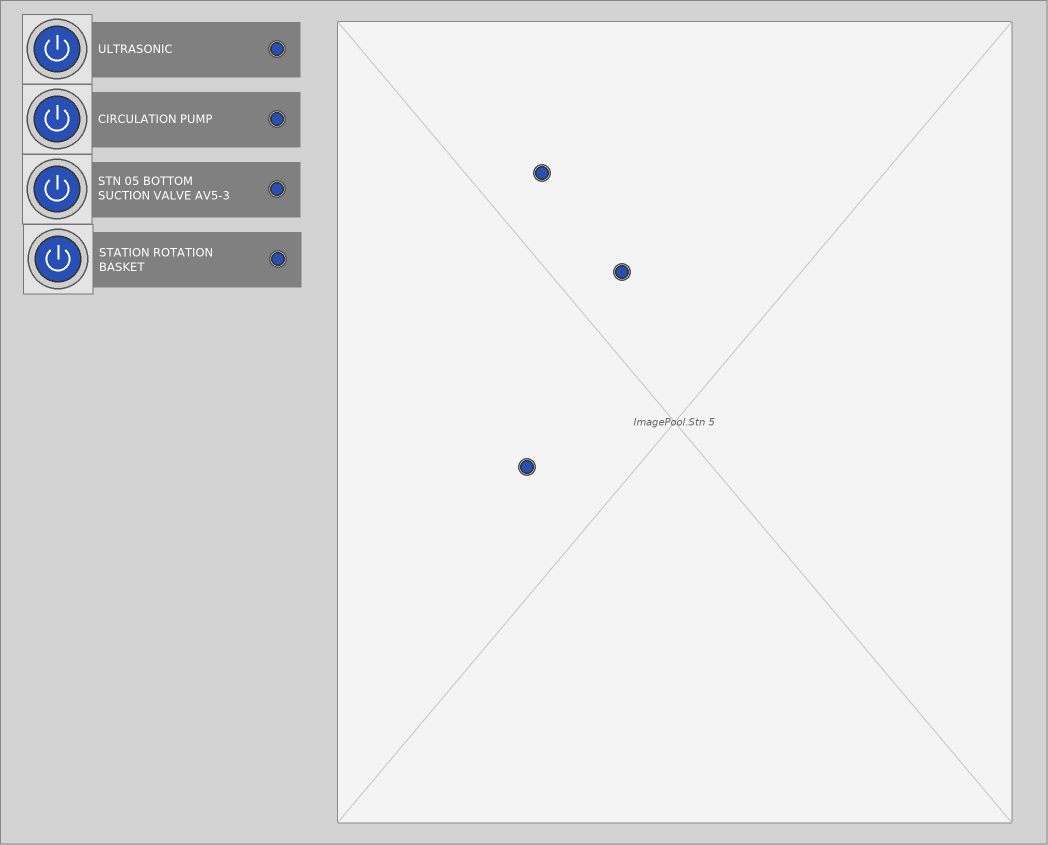
VISUALIZATION Recipe_Station05  // 1048x845
    Rectangle (0,0 1048x845)
    Image (337,21 675x802), image: ImagePool.Stn 5
    RoundedRectangle (61,22 239x55)
    Label (95,41 163x16), "ULTRASONIC"
    Lamp1 (267,39 20x20), variable: DSScrMapSSUR.DsSubRecipeMemory.bOut3EnProTankBottomUltrasonicA, style: Lamp-Lamp1-Blue
    PowerSwitch (22,14 70x70), variable: DSScrMapSSUR.DsSubRecipeMemory.bOut3EnProTankBottomUltrasonicA, behaviour: TOGGLE, style: Switch-PowerSwitch-Blue
    RoundedRectangle (69,92 231x55)
    Label (95,111 151x16), "CIRCULATION PUMP"
    Lamp1 (267,109 20x20), variable: DSScrMapSSUR.DsSubRecipeMemory.bOut1EnProTankPump, style: Lamp-Lamp1-Blue
    PowerSwitch (22,84 70x70), variable: DSScrMapSSUR.DsSubRecipeMemory.bOut1EnProTankPump, behaviour: TOGGLE, style: Switch-PowerSwitch-Blue
    RoundedRectangle (69,162 231x55)
    Label (95,174 151x29), "STN 05 BOTTOM SUCTION VALVE AV5-3"
    Lamp1 (267,179 20x20), variable: DSScrMapSSUR.DsSubRecipeMemory.bOut3ActValve3, style: Lamp-Lamp1-Blue
    PowerSwitch (22,154 70x70), variable: DSScrMapSSUR.DsSubRecipeMemory.bOut3ActValve3, behaviour: TOGGLE, style: Switch-PowerSwitch-Blue
    Lamp1 (532,163 20x20), variable: DSScrMapSSUR.DsSubRecipeMemory.bOut3EnProTankBottomUltrasonicA, style: Lamp-Lamp1-Blue
    Lamp1 (517,457 20x20), variable: DSScrMapSSUR.DsSubRecipeMemory.bOut1EnProTankPump, style: Lamp-Lamp1-Blue
    Lamp1 (612,262 20x20), variable: DSScrMapSSUR.DsSubRecipeMemory.bOut3ActValve3, style: Lamp-Lamp1-Blue
    RoundedRectangle (70,232 231x55)
    Label (96,245 151x30), "STATION ROTATION BASKET"
    Lamp1 (268,249 20x20), variable: DSScrMapSSUR.DsSubRecipeMemory.bOut14EnInstrument3, style: Lamp-Lamp1-Blue
    PowerSwitch (23,224 70x70), variable: DSScrMapSSUR.DsSubRecipeMemory.bOut14EnInstrument3, behaviour: TOGGLE, style: Switch-PowerSwitch-Blue
END_VISUALIZATION

(* stored: Version 1.1.0.1, ProductVersion 3.1.4024.12
   Visu Recipe_Station05: Id {5a5ab2ef-40ad-4c73-9ee9-fe339858362a} *)
